TEXTLIST E_FaultTypes
  0 = 'NA'
  1 = 'OM'
  2 = 'MC'
  3 = 'CF'
  4 = 'FF'
   = ''
END_TEXTLIST

(* stored: Version 1.1.0.1, ProductVersion 3.1.4024.3
   TextList E_FaultTypes: Id {3024e051-382d-4c75-9c0d-238f7f237aaa} *)
